(* IEC 61131-3 sources: AxTestProject/Program/LStandardLibrary/Signal Handling, 7 files *)

(* ---- AnalogSignal.st ---- *)
NAMESPACE stdLib.SignalHandling
    CLASS AnalogSignal

        VAR PRIVATE
            m_status : AnalogSignalStatus;
            m_Old : BOOL;
            m_minValue : LREAL;
            m_maxValue : LREAL;
        END_VAR

        //##################################################################
        // Method EnableLimiter
        //
        // Enables limitation for analog signal. If limitation enabled,
        // the status bits "MinLimitReached" and "MaxLimitReached" will be
        // set, if the signal exceeds the limits.
        //
        // min : minimal limitation
        // max : max limitation
        //##################################################################
        METHOD PUBLIC EnableLimiter
            VAR_INPUT
                min : LREAL;
                max : LREAL;
            END_VAR
            m_minValue := min;
            m_maxValue := max;
            m_Status.LimiterIsEnabled := TRUE;
        END_METHOD

        //##################################################################
        // Method DisableLimiter
        //
        // Disables limitation for analog signal. If limitation disabled,
        // the status bits "MinLimitReached" and "MaxLimitReached" will not
        // set, if the signal exceeds the limits.
        //##################################################################
        METHOD PUBLIC DisableLimiter
            m_Status.LimiterIsEnabled := FALSE;
        END_METHOD

        //##################################################################
        // Method execute
        //
        // Executes the signal evaluation
        //
        // Parameter:
        // signal : The analog signal to be evaluated
        // enable : Enables the signal evaluation
        // qDefault : Default value, if enable = false
        // Norm : Nomalize factor for signal
        //##################################################################
        METHOD PUBLIC execute : AnalogSignalStatus
            VAR_INPUT
                signal : LREAL;
                enable : BOOL := TRUE;
                qDefault : LREAL := 0.0;
                Norm : LREAL := LREAL#1.0;
            END_VAR
            VAR_TEMP
                actValue : LREAL;
            END_VAR
            IF (enable) THEN
                actValue := signal;
                m_status.QBAD := FALSE;
            ELSE
                actValue := qDefault;
                m_status.QBAD := TRUE;
            END_IF;

            // Check Limits if enabled
            IF (m_Status.LimiterIsEnabled) THEN
                m_status.MaxLimitReached := (actValue >= m_maxValue);
                m_status.MinLimitReached := (actValue <= m_minValue);
            ELSE
                m_status.MaxLimitReached := FALSE;
                m_status.MinLimitReached := FALSE;
            END_IF;

            IF (m_status.MaxLimitReached) THEN
                m_status.Q := m_maxValue;
            ELSIF (m_status.MinLimitReached) THEN
                m_status.Q := m_minValue;
            ELSE
                m_status.Q := actValue;
            END_IF;

            execute := m_status;

        END_METHOD

    END_CLASS

    TYPE AnalogSignalStatus : STRUCT
            Q : LREAL;
            QBad : BOOL;
            MaxLimitReached : BOOL;
            MinLimitReached : BOOL;
            LimiterIsEnabled : BOOL := FALSE;
        END_STRUCT;
    END_TYPE

END_NAMESPACE

(* ---- BinSignal.st ---- *)
NAMESPACE stdLib.SignalHandling
    CLASS BinSignal

        VAR PRIVATE
            m_status : BinSignalStatus;
            m_Old : BOOL;
        END_VAR

        METHOD PUBLIC execute : BinSignalStatus
            VAR_INPUT
                signal : BOOL;
                enable : BOOL := TRUE;
                qDefault : BOOL := FALSE;
            END_VAR
            VAR_TEMP
                sig : BOOL;
            END_VAR
            IF (enable) THEN
                sig := signal;
                m_status.QBAD := FALSE;
            ELSE
                sig := qDefault;
                m_status.QBAD := TRUE;
            END_IF;

            m_Status.QRis := sig AND NOT(m_Old);
            m_Status.QFal := NOT(sig) AND m_Old;
            m_Old := sig;
            m_status.Q := sig;

            execute := m_status;
        END_METHOD

    END_CLASS

    TYPE BinSignalStatus : STRUCT
            Q : BOOL;
            QRis : BOOL;
            QFal : BOOL;
            QBad : BOOL;
        END_STRUCT;
    END_TYPE

END_NAMESPACE

(* ---- Encoder.st ---- *)
NAMESPACE stdLib.SignalHandling
    CLASS Encoder
        VAR PRIVATE
            m_aOld : BOOL;
            m_bOld : BOOL;
            m_status : EncoderStatus;
        END_VAR

        // Reset encoder position to zero
        METHOD PUBLIC Reset
            m_status.position := DINT#0;
        END_METHOD

        //Set encoder to specific position
        METHOD PUBLIC Set
            VAR_INPUT
                position : DINT;
            END_VAR
                m_Status.position := position;
                ;
        END_METHOD

        //Evaluate encoder signals A and B
        METHOD PUBLIC evaluate
            VAR_INPUT
                a : BOOL;
                b : BOOL;
            END_VAR
            VAR_TEMP
                aRis : BOOL;
                bRis : BOOL;
                aFal : BOOL;
                bFal : BOOL;
            END_VAR

            aRis := a AND NOT(m_aOld);
            aFal := NOT(a) AND m_aOld;
            m_aOld := a;

            bRis := b AND NOT(m_bOld);
            bFal := NOT(b) AND m_bOld;
            m_bOld := b;

            //Forward detection
            IF (
                aRis AND NOT(b)
                OR a AND bRis
                OR aFal AND b
                OR NOT(a) AND bFal) THEN
                m_status.isInMotion := true;
                m_status.direction := false;
                m_status.position := m_status.position + DINT#1;
                m_status.increments := m_status.increments + DINT#1;
            //Reverse detection
            ELSIF
            (
                aRis AND b
                OR NOT(a) AND bRis
                OR aFal AND NOT(b)
                OR a AND bFal) THEN
                m_status.isInMotion := true;
                m_status.direction := true;
                m_status.position := m_status.position - DINT#1;
                m_status.increments := m_status.increments - DINT#1;
            ELSE
                m_status.isInMotion := false;
                m_status.direction := false;
            END_IF;

        END_METHOD

        METHOD PUBLIC GetStatus : EncoderStatus
            ;
            GetStatus := m_status;
            m_status.increments := DINT#0;
        END_METHOD

        METHOD PUBLIC SetInternals
            VAR_INPUT
                aOld : BOOL;
                bOld : BOOL;
            END_VAR
            m_aOld := aOld;
            m_bOld := bOld;
        END_METHOD

    END_CLASS

    TYPE EncoderStatus :
        STRUCT
            position : DINT;  // increments since last reset
            increments : DINT; // increments since last GetStatus-Call
            direction : BOOL; // 0: forward; 1: reverse
            isInMotion : BOOL; // encoder is in motion
        END_STRUCT;
    END_TYPE
END_NAMESPACE

(* ---- OnDelay.st ---- *)
NAMESPACE stdLib.Timer
    CLASS OnDelay
        VAR
            m_timeElapsed : INT;
            m_status : Timerstatus;
            m_old : BOOL;
            m_isRunning : BOOL;
            m_PT : INT;
        END_VAR

        METHOD Start
            VAR_INPUT
                PT : INT;
                Retrigger : BOOL := false;
            END_VAR
            VAR_TEMP
            END_VAR
                if (retrigger OR NOT(m_isRunning)) THEN
                    m_PT := PT;
                    m_status.ET := m_PT;
                    m_isRunning := true;
                END_IF;
        END_METHOD

        METHOD Execute : BOOL
            VAR_INPUT
            END_VAR
            VAR_TEMP
                tQ : BOOL;
            END_VAR

            if (m_status.ET > m_PT) then
                m_status.ET := m_status.ET - 1;
            end_if;

            if (m_status.ET <= m_PT) then
                tQ := true;
                m_isRunning := false;
            ELSE
                tQ := false;
            END_IF;
            m_status.Q := tQ;
            Execute := tQ;
        END_METHOD

        METHOD Q : BOOL
            VAR_INPUT
            END_VAR
            VAR_TEMP
            END_VAR
            Q := m_status.Q;
                ;
        END_METHOD

        METHOD GetStatus : Timerstatus
            VAR_INPUT
            END_VAR
            VAR_TEMP
            END_VAR
                GetStatus := m_status;
                ;
        END_METHOD

    END_CLASS

    TYPE Timerstatus :
        STRUCT
            Q : BOOL;
            ET : INT;
        END_STRUCT;
    END_TYPE

END_NAMESPACE

(* ---- BinSignalTest.st ---- *)
NAMESPACE StdLibTesting.BinSignal

    {Test(iSignal := 0, iEnable := 0, iDefault := 0, iExpQ := 0, iExpQBad := 1)}
    {Test(iSignal := 0, iEnable := 0, iDefault := 1, iExpQ := 1, iExpQBad := 1)}
    {Test(iSignal := 0, iEnable := 1, iDefault := 0, iExpQ := 0, iExpQBad := 0)}
    {Test(iSignal := 0, iEnable := 1, iDefault := 1, iExpQ := 0, iExpQBad := 0)}

    {Test(iSignal := 1, iEnable := 0, iDefault := 0, iExpQ := 0, iExpQBad := 1)}
    {Test(iSignal := 1, iEnable := 0, iDefault := 1, iExpQ := 1, iExpQBad := 1)}
    {Test(iSignal := 1, iEnable := 1, iDefault := 0, iExpQ := 1, iExpQBad := 0)}
    {Test(iSignal := 1, iEnable := 1, iDefault := 1, iExpQ := 1, iExpQBad := 0)}

    FUNCTION execute
        VAR_INPUT
            iSignal : INT;
            iEnable : INT;
            iDefault : INT;
            iExpQ : INT;
            iExpQBad : INT;
        END_VAR

        VAR_TEMP
            o : stdLib.SignalHandling.BinSignal;
            status : stdLib.SignalHandling.BinSignalStatus;
            tSignal : BOOL;
            tEnable : BOOL;
            tDefault : BOOL;
            tExpQ : BOOL;
            tExpQBad : BOOL;
        END_VAR

        tSignal := iSignal <> 0;
        tEnable := iEnable <> 0;
        tDefault := iDefault <> 0;
        tExpQ := iExpQ <> 0;
        tExpQBad := iExpQBad <> 0;

        status := o.execute(signal := tSignal, enable := tEnable, qDefault := tDefault);
        Assert_Equal_BOOL(expected := tExpQ, actual := status.Q);
        ;
            ;
    END_FUNCTION

    {Test(iSignal := 1, iEnable := 1, iDefault := 0, iExpQ := 1, iExpQRis := 1, iExpQFal := 0, iTestFallingEdge := 0)}
    {Test(iSignal := 0, iEnable := 1, iDefault := 0, iExpQ := 0, iExpQRis := 0, iExpQFal := 1, iTestFallingEdge := 1)}

    FUNCTION QRis
        VAR_INPUT
            iSignal : INT;
            iEnable : INT;
            iDefault : INT;
            iExpQ : INT;
            iExpQRis : INT;
            iExpQFal : INT;
            iTestFallingEdge : INT;
        END_VAR
        VAR_TEMP
            o : stdLib.SignalHandling.BinSignal;
            status : stdLib.SignalHandling.BinSignalStatus;
            tSignal : BOOL;
            tEnable : BOOL;
            tDefault : BOOL;
            tExpQ : BOOL;
            tExpQRis : BOOL;
            tExpQFal : BOOL;
            tTestFallingEdge : BOOL;
        END_VAR

        tSignal := iSignal <> 0;
        tEnable := iEnable <> 0;
        tDefault := iDefault <> 0;
        tExpQ := iExpQ <> 0;
        tExpQRis := iExpQRis <> 0;
        tExpQFal := iExpQFal <> 0;
        tTestFallingEdge := iTestFallingEdge <> 0;

        if (tTestFallingEdge) then
            status := o.execute(signal := true, enable := tEnable, qDefault := tDefault);
        END_IF;

        status := o.execute(signal := tSignal, enable := tEnable, qDefault := tDefault);
        Assert_Equal_BOOL(expected := tExpQ, actual := status.Q);
        Assert_Equal_BOOL(expected := tExpQRis, actual := status.QRis);
        Assert_Equal_BOOL(expected := tExpQFal, actual := status.QFal);

        status := o.execute(signal := tSignal, enable := tEnable, qDefault := tDefault);
        Assert_Equal_BOOL(expected := tExpQ, actual := status.Q);
        Assert_Equal_BOOL(expected := false, actual := status.QRis);
        Assert_Equal_BOOL(expected := false, actual := status.QFal);
    END_FUNCTION
END_NAMESPACE

(* ---- EncoderTest.st ---- *)
NAMESPACE StdLibTesting.Encoder

    {Test}
    FUNCTION Reset
        VAR_INPUT
        END_VAR
        VAR_TEMP
            o : stdLib.SignalHandling.Encoder;
            status : stdLib.SignalHandling.EncoderStatus;
        END_VAR

        o.Set(DINT#555);
        status := o.GetStatus();
        Assert_Equal_DINT(expected := DINT#555, actual := status.position);
        o.Reset();
        status := o.GetStatus();
        Assert_Equal_DINT(expected := DINT#0, actual := status.position);
        Assert_Equal_DINT(expected := DINT#0, actual := status.increments);
        ;
            ;
    END_FUNCTION

    {Test( aOld := 0, a := 0, bOld := 0, b := 0, dir := 0, pos := 0)}
    {Test( aOld := 1, a := 1, bOld := 1, b := 1, dir := 0, pos := 0)}

    {Test( aOld := 0, a := 1, bOld := 0, b := 0, dir := 0, pos := 1)}
    {Test( aOld := 1, a := 0, bOld := 1, b := 1, dir := 0, pos := 1)}
    {Test( aOld := 1, a := 1, bOld := 0, b := 1, dir := 0, pos := 1)}
    {Test( aOld := 0, a := 0, bOld := 1, b := 0, dir := 0, pos := 1)}

    {Test(a := 1, b := 1, aOld := 0, bOld := 1, dir := 1, pos := -1)}
    {Test(a := 0, b := 1, aOld := 0, bOld := 0, dir := 1, pos := -1)}
    {Test(a := 0, b := 0, aOld := 1, bOld := 0, dir := 1, pos := -1)}
    {Test(a := 1, b := 0, aOld := 1, bOld := 1, dir := 1, pos := -1)}

    FUNCTION EncoderDirection
        VAR_INPUT
            a : INT;
            b : INT;
            aOld : INT;
            bOld : INT;
            dir : INT;
            pos : INT;
        END_VAR
        VAR
            tA : BOOL;
            tB : BOOL;
            tAOld : BOOL;
            tBOld : BOOL;
            tDir : BOOL;
            o : stdLib.SignalHandling.Encoder;
            status : stdLib.SignalHandling.EncoderStatus;
        END_VAR
        tA := a <> 0;
        tB := b <> 0;
        tAOld := aOld <> 0;
        tBold := bOld <> 0;
        tDir := dir <> 0;
        o.SetInternals(aOld := tAOld, bOld:= tBold);
        o.Evaluate(tA, tB);
        status := o.GetStatus();

        Assert_Equal_BOOL(expected := tDir, actual := status.direction);
        Assert_Equal_DINT(expected := INT_TO_DINT(pos), actual := status.position);
        Assert_Equal_DINT(expected := INT_TO_DINT(pos), actual := status.increments);

        status := o.GetStatus();
        Assert_Equal_DINT(expected := INT_TO_DINT(pos), actual := status.position);
        Assert_Equal_DINT(expected := DINT#0, actual := status.increments);
        ;
    END_FUNCTION
END_NAMESPACE

(* ---- ClockGenerator.st ---- *)
NAMESPACE stdLib.Timer
    CLASS ClockGenerator

    VAR PRIVATE
        m_timer1 : OnDelay;
        m_timer2 : OnDelay;
        m_isRunning : BOOL;
        m_q : BOOL;
    END_VAR

    METHOD PUBLIC Execute
        VAR_INPUT
            pulse : DINT;
            pause : DINT;
            sysLibTimer : DINT;
        END_VAR

            m_timer1.Execute(sysLibTimer);
            m_timer2.Execute(sysLibTimer);

            IF (m_timer2.Q() OR not(m_isRunning)) THEN
                m_timer1.Start(PT := pulse);
                m_timer2.Reset();
                m_isRunning := true;
                m_q := true;
            END_IF;

            if (m_timer1.Q() ) then
                m_timer2.Start(PT:=pause);
                m_timer1.Reset();
                m_q := false;
            End_if;
    END_METHOD

    METHOD PUBLIC Q : BOOL
        Q := m_q;
    END_METHOD

    END_CLASS

END_NAMESPACE
